(* IEC 61131-3 sources: eCockpitGit/test_project/src/%F%00 Library/%F%Common Functions/%F%String/%F%Normal, 1 file *)

(* ---- %POU%FU_CheckNumber.st ---- *)
//This function checks if a string only contains numbers, dot (.) and dash (-) are also permitted as they are required for some numbers
//Returns true if string only contains numbers
// |**Version**|**Author**| **Date** |**Changes**
// | 1         | NSN      | 10-12-18 | Creation
FUNCTION FU_CheckNumber : BOOL
VAR_INPUT
	str			:STRING(255);	//String
END_VAR
(*%!%__DELIMITER__%!%*)
FU_CheckNumber		:=		FU_CheckNumberBI(str:=str);
